// TIA Portal V16 export
// export: Created 2021-02-18T15:18:45.231461Z, ExportSetting WithDefaults, DisplayName Totally Integrated Automation Portal, DisplayVersion V16 Update 3, DisplayName TIA Portal Version Control Interface, DisplayVersion V16 Update 2, DisplayName TIA Portal Openness, DisplayVersion V16 Update 3, DisplayName STEP 7 Professional, DisplayVersion V16 Update 3, DisplayName STEP 7 Safety, DisplayVersion V16, DisplayName WinCC Professional, DisplayVersion V16 Update 3
TYPE "UT01000_St_SysRevision"
TITLE = Static UDT — Sys - Revision Data
// Revision Data
// stored: IsFailsafeCompliant false
   STRUCT
      REV_BLOCK { ExternalWritable := 'False'; S7_SetPoint := 'True'} : String[7];   // Block or Project number
      REV_NUMBER { ExternalWritable := 'False'; S7_SetPoint := 'True'} : String[20];   // Revision status followed by revision number
      REV_DATE { ExternalWritable := 'False'; S7_SetPoint := 'True'} : String[10];   // Revision date
      REV_AUTHOR { ExternalWritable := 'False'; S7_SetPoint := 'True'} : String[20];   // Revision author
   END_STRUCT;
END_TYPE
